//{attribute 'qualified_only'}
//{attribute 'strict'}
TYPE E_RecipeMode :
(
	eRecipeMode_None := 0,
	eRecipeMode_ToFrom,
	
	eRecipeMode_Max
);
END_TYPE

(* stored: Version 1.1.0.1
   EnumerationTextList E_RecipeMode: Id {65cdb34a-288d-4211-b848-df62c007bf3e} *)
